TYPE tstCTCStatusBits :
STRUCT
	TrackingErrorToleranceExceeded 	:BOOL;
	WarningActive					:BOOL;
	MotionModeActive				:BOOL;
	MotionCommandCompleted 			:BOOL;	
	LimitSwitchIn					:BOOL;	
	LimitSwitchOut					:BOOL;
	Homed							:BOOL;
	Ready							:BOOL;
END_STRUCT
END_TYPE

(* stored: Version 1.1.0.1, ProductVersion 3.1.4026.17
   DUT tstCTCStatusBits: Id {ff28900c-8d4b-4409-b2d1-d07fdb089f3b} *)
